{attribute 'GeneratedUsingTerminal: EJ1957-0000-0017'}
{attribute addProperty BoxType "EJ1957-0000-0017"}
{attribute addProperty Id "FSoE_InputsFSoE_Inputs_8A5FBAF818FSoE_OutputsFSoE_Outputs_1F40D10314"}
{attribute addProperty CRC "2680868372"}
{attribute addProperty Size "32"}
TYPE Module_1_FSOE_9FCACE14 :
STRUCT
	{attribute addProperty Name "FSoE_Inputs"}
	FSoE_Inputs  : FSoE_Inputs_8A5FBAF8;
	{attribute addProperty Name "FSoE_Outputs"}
	FSoE_Outputs  : FSoE_Outputs_1F40D103;
END_STRUCT
END_TYPE

(* stored: Version 1.2.0.0, ProductVersion 3.1.4024.9
   DUT Module_1_FSOE_9FCACE14: Id {47c9de10-cbe6-4103-99a0-56ad14454d69} *)
